// TIA Portal V15.1 export
// export: Created 2024-06-21T08:41:08.753447Z, ExportSetting WithDefaults, DisplayName Totally Integrated Automation Portal, DisplayVersion V15.1 Update 5, DisplayName TIA Portal Openness, DisplayVersion V15.1 Update 5, DisplayName SINAMICS Startdrive Advanced, DisplayVersion V15.1, DisplayName G130, G150, S120, S150, SINAMICS MV, S210, DisplayVersion V15.1, DisplayName G110M, G120, G120C, G120D, G120P, DisplayVersion V15.1, DisplayName STEP 7 Professional, DisplayVersion V15.1 Update 5, DisplayName STEP 7 Safety, DisplayVersion V15.1, DisplayName WinCC Professional, DisplayVersion V15.1 Update 5, DisplayName SIMATIC Visualization Architect, DisplayVersion V15.1
FUNCTION "LGBCrossConvIAnim" : Void   // FC6632, FBD
TITLE = LIAnimDWord / LGBCrossConvIAnim
{ S7_Optimized_Access := 'TRUE' }
AUTHOR : VCC
FAMILY : Anim
NAME : SIAnim
VERSION : 0.1
// =============================================================================
// Handles the conversion from bits to one Word for simple icon Animation. 
// =============================================================================
// stored: AutoNumber false, IsIECCheckEnabled false, SetENOAutomatically False, UDAEnableTagReadback false
   VAR_INPUT
      I_Active : Bool;   // Active
      I_AutoMode : Bool;   // Auto mode
      I_AutoModeSel : Bool;   // Auto selected
      I_ManualMode : Bool;   // Manual mode / Manual Mode
      I_ManualModeSel : Bool;   // Manual selected
      I_ManSetIntlk : Bool;   // Manual motor Set interlock
      I_ManResIntlk : Bool;   // Manual motor Res interlock
      I_SafetyOk : Bool;   // Safety Ok
      I_MotionStopOk : Bool;   // Service Active / Motion stop Ok
      I_FncSelInHMI : Bool;   // Manual selection from HMI
   END_VAR
   VAR_OUTPUT
      H_IAnim : DWord;   // Icon animation Word / Icon Animation
   END_VAR
BEGIN

REGION Network 1: **** 1 - Inputs **** Active
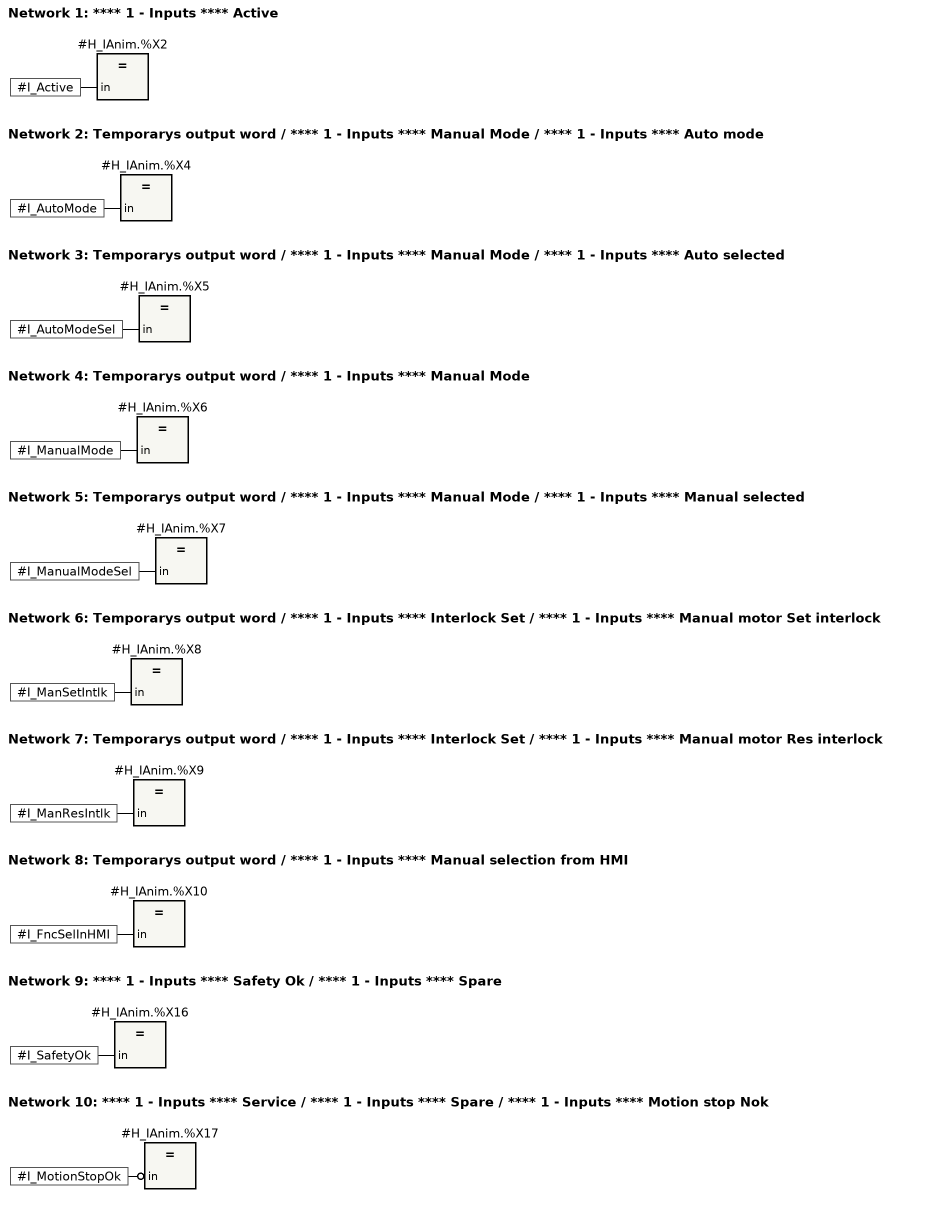
   #H_IAnim.%X2 := #I_Active;
END_REGION

REGION Network 2: Temporarys output word / **** 1 - Inputs **** Manual Mode / **** 1 - Inputs **** Auto mode
   // Manual Mode
   #H_IAnim.%X4 := #I_AutoMode;
END_REGION

REGION Network 3: Temporarys output word / **** 1 - Inputs **** Manual Mode / **** 1 - Inputs **** Auto selected
   // Manual Mode
   #H_IAnim.%X5 := #I_AutoModeSel;
END_REGION

REGION Network 4: Temporarys output word / **** 1 - Inputs **** Manual Mode
   // Manual Mode
   #H_IAnim.%X6 := #I_ManualMode;
END_REGION

REGION Network 5: Temporarys output word / **** 1 - Inputs **** Manual Mode / **** 1 - Inputs **** Manual selected
   // Manual Mode
   #H_IAnim.%X7 := #I_ManualModeSel;
END_REGION

REGION Network 6: Temporarys output word / **** 1 - Inputs **** Interlock Set / **** 1 - Inputs **** Manual motor Set interlock
   // Interlock Set
   #H_IAnim.%X8 := #I_ManSetIntlk;
END_REGION

REGION Network 7: Temporarys output word / **** 1 - Inputs **** Interlock Set / **** 1 - Inputs **** Manual motor Res interlock
   // Interlock Set
   #H_IAnim.%X9 := #I_ManResIntlk;
END_REGION

REGION Network 8: Temporarys output word / **** 1 - Inputs **** Manual selection from HMI
   // Manual selection from HMI
   #H_IAnim.%X10 := #I_FncSelInHMI;
END_REGION

REGION Network 9: **** 1 - Inputs **** Safety Ok / **** 1 - Inputs **** Spare
   // Safety Ok / Spare
   #H_IAnim.%X16 := #I_SafetyOk;
END_REGION

REGION Network 10: **** 1 - Inputs **** Service / **** 1 - Inputs **** Spare / **** 1 - Inputs **** Motion stop Nok
   // Service / Spare / Motion stop NOK
   #H_IAnim.%X17 := NOT #I_MotionStopOk;
END_REGION
END_FUNCTION
